PROGRAM SqlDbReadWrite
VAR_OUTPUT
	ready : BOOL;
END_VAR
VAR
	fbSQLCommand : FB_SQLCommandEvt(sNetID := '', tTimeout := T#5S);
	fbSQLDatabase : FB_SQLDatabaseEvt (sNetID := '', tTimeout := T#5S);
	fbSQLResult : FB_SQLResultEvt(sNetID:='', tTimeout:=T#5S);
	
	query : STRING(1000);
	step : DatabaseStep;
	
	cachedBuffer : ARRAY[0..100000] OF BYTE;
END_VAR

IF NOT ready THEN
	setup();
	RETURN;
END_IF

CASE step OF
	DatabaseStep.IDLE:
		IF fbSQLDatabase.CreateCmd(ADR(fbSQLCommand)) THEN
			step := DatabaseStep.EXECUTE;
		END_IF
		
	DatabaseStep.EXECUTE:
		IF fbSQLCommand.ExecuteDataReturn(ADR(query), SIZEOF(query), ADR(fbSqlResult)) THEN
			query := '';
			step := DatabaseStep.LOAD_DATA;
		END_IF
		
	DatabaseStep.LOAD_DATA:
		fbSqlResult.Read(
			nStartIndex := 0,
			nRecordCount := 1,
			pData := ADR(cachedBuffer),
			cbData := SIZEOF(cachedBuffer),
			bWithVerifying := FALSE,
			bDataRelease := FALSE);
			
END_CASE

METHOD execute : BOOL
VAR_INPUT
	queryInstruction : STRING(1000);
END_VAR
query := queryInstruction;
END_METHOD

METHOD reset : BOOL
VAR_INPUT
END_VAR
step := RESET;
END_METHOD

METHOD setup : BOOL
CASE step OF
	DatabaseStep.RESET:
		step := DatabaseStep.DISCONNECT;
		
	DatabaseStep.CONNECT:
		IF fbSQLDatabase.Connect(1) THEN
			IF NOT fbSqlDatabase.bError THEN
				step := DatabaseStep.IDLE;
				setup := TRUE;
			END_IF
		END_IF
		
	DatabaseStep.DISCONNECT:
		IF fbSQLDatabase.Disconnect() THEN
			step := DatabaseStep.CONNECT;
		END_IF
END_CASE
END_METHOD

END_PROGRAM

(* stored: Version 1.1.0.1, ProductVersion 3.1.4024.11
   POU SqlDbReadWrite: Id {0bc2a762-06ca-483c-b0e0-dd7ad2baba5d}, SpecialFunc None
   Method execute: Id {ed26c3db-5f41-471b-b73a-a72f1a0a0427}
   Method reset: Id {822ca499-73a6-4858-9847-01a0c485f426}
   Method setup: Id {a18eda8a-807b-45f9-98ea-29ab8720a940} *)
